(* IEC 61131-3 sources: WebSocketBenchmark/programSt/pous/programs, 1 file *)

(* ---- main.st ---- *)
PROGRAM main
VAR
	output : int AT %MW0 := 0;
END_VAR

output := output + 1;

END_PROGRAM
